PROGRAM P_BACnet_Scene
VAR
END_VAR

//keep BACnet object alive
fbBACnet_AV_SL_Scene(Device := Device, bEnablePV := TRUE, bNullPV := FALSE);

END_PROGRAM

(* stored: Version 1.1.0.1, ProductVersion 3.1.4024.5
   POU P_BACnet_Scene: Id {f07e323b-ee39-43cc-a08a-3a2180e8598f}, SpecialFunc None *)
